// TIA Portal V18 export
TYPE "LGasp_flyingCutoff"
// stored: IsFailsafeCompliant false
   STRUCT
      state : Struct
         automatic : Bool;   // taglio in automatico
         fault : Bool;   // asse taglio al volo in errore
         fcpos : Bool;   // fine corsa positivo
         fcneg : Bool;   // fine corsa negatico
         sync : Bool;   // carro al volo sincronizzato
         home : Bool;   // carro al volo in posizione di home
         programvalid : Bool;   // programma SMC valido
         posok : Bool;   // motore in posizione ok
      END_STRUCT;
      RM_position : Real;   // posizione ruota metrica in mm (visualizzazione)
      motor_position : Real;   // posizione motore in mm (visualizzazione)
      cutlength : Real;   // VFR600 lunghezza di taglio (visualizzazione)
      maskwindow : Real;   // VFR601 oscuramento (visualizzazione)
      cutoffset : Real;   // VFR602 offset di taglio (visualizzazione)
      numLaser : Real;   // numero di laser di sincronismo presenti, serve al PC per visualizzare quelli presenti
      lengthdone : Real;   // Lunghezza tagliata VS125 (visualizzazione)
      enableChangeLaser : Bool;   // 1= abilitazione cambio laser
      laser1 : Struct
         "name" : WString;   // etichetta laser
         enable : Bool;   // laser abilitato da pagina del supervisore
         stateON : Bool;   // stato (per avere lo stato di I.A1.X31.Pin4 inserire le istruzione nel programma SMC come fatto per gli extracorsa)
      END_STRUCT;
      laser2 : Struct
         "name" : WString;   // etichetta laser
         enable : Bool;   // laser abilitato da pagina del supervisore
         stateON : Bool;   // stato (per avere lo stato di I.A1.X31.Pin4 inserire le istruzione nel programma SMC come fatto per gli extracorsa)
      END_STRUCT;
      laser3 : Struct
         "name" : WString;   // etichetta laser
         enable : Bool;   // laser abilitato da pagina del supervisore
         stateON : Bool;   // stato (per avere lo stato di I.A1.X31.Pin4 inserire le istruzione nel programma SMC come fatto per gli extracorsa)
      END_STRUCT;
      numpos : Int;   // numero di posizioni di cambio stampo 1..4 home escluso
      poshome : Struct   // finestra di tolleranza posizione valvola in quota [mm]
         start : Bool;   // 1= pulsante premuto start asse taglio in posizione
         limitemin : LReal;   // da PLC
         limitemax : LReal := 1000.0;   // da PLC
         valore : LReal;   // da programma PC
      END_STRUCT;
      pos : Array[1..4] of Struct   // posizioni magazzino cambio stampi
         start : Bool;   // 1= pulsante premuto start asse taglio in posizione
         limitemin : LReal;   // da PLC
         limitemax : LReal;   // da PLC
         valore : LReal;   // da programma PC
      END_STRUCT;
   END_STRUCT;
   // pos[1].limitemax := 1000.0;
END_TYPE
